TYPE ST_Palette :
STRUCT
	PaletteDimensionX : INT;
	PaletteDimensionY : INT;
	
	ActualPalettePositionX : INT;
	ActualPalettePositionY : INT;
END_STRUCT
END_TYPE

(* stored: Version 1.1.0.1, ProductVersion 3.1.4020.12
   DUT ST_Palette: Id {16326acd-ff40-45ea-bade-89e0095759d1} *)
